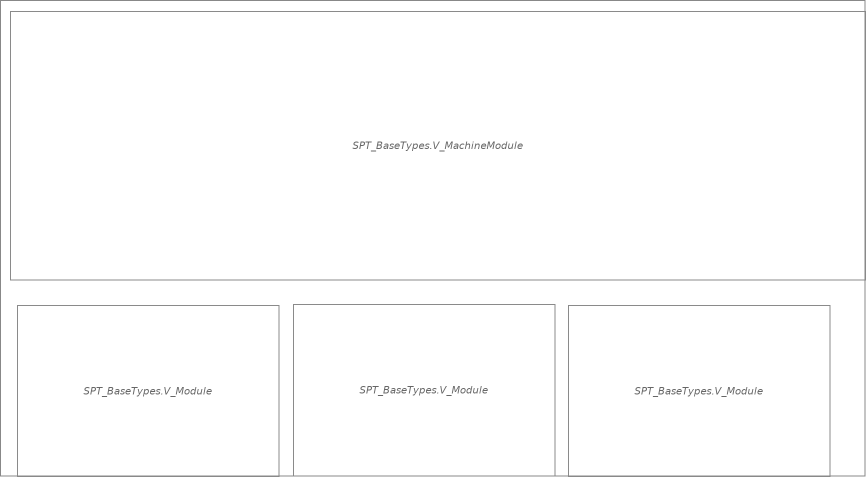
VISUALIZATION Visualization  // 866x477
    Frame (10,11 856x269)
        shows SPT_BaseTypes.V_MachineModule(HMI := MAIN.Machine.PackMLBaseModule_HMI)
    Frame (17,305 262x172)
        shows SPT_BaseTypes.V_Module(HMI := MAIN.Machine.Infeed.PackMLBaseModule_HMI)
    Frame (293,304 262x172)
        shows SPT_BaseTypes.V_Module(HMI := MAIN.Machine.Process.PackMLBaseModule_HMI)
    Frame (568,305 262x172)
        shows SPT_BaseTypes.V_Module(HMI := MAIN.Machine.Outfeed.PackMLBaseModule_HMI)
END_VISUALIZATION

(* stored: Version 1.1.0.1, ProductVersion 3.1.4024.12
   Visu Visualization: Id {afee2981-84b8-4371-8ffe-1a9005db9bad} *)
